{attribute 'call_after_init'}
FUNCTION_BLOCK A EXTENDS Object
VAR_INPUT
END_VAR
VAR_OUTPUT
END_VAR
VAR
	B1: B;
	C1: C;
	tT: BoolParam;
	tU: UdintParam;
	tR: RealParam;
END_VAR

END_FUNCTION_BLOCK

(* stored: Version 1.1.0.1, ProductVersion 3.1.4024.12
   POU A: Id {6af5d0de-e557-45e7-9f62-300c51773914}, SpecialFunc None *)
